DATA_BLOCK "ST10_MaterialGate6_DB"
{ S7_Optimized_Access := 'FALSE' }
VERSION : 0.1
NON_RETAIN
"SafetyGate"

BEGIN

END_DATA_BLOCK

